Fanuc KAREL source: KO00014.KL

PROGRAM KO00014
%NOLOCKGROUP
VAR
  P1: XYZWPR
  P2: XYZWPR
  P3: XYZWPR
  P4: XYZWPR
  OUT: XYZWPR
BEGIN
  OUT = FRAME(P1, P2, P3, P4)
END KO00014
